(* CoDeSys 2.3 export: CRC16.EXP *)

(* Data type in INT *)
TYPE CRC16 : UINT;
END_TYPE
